(* IEC 61131-3 sources: CodesysTest/export/Function Blocks/SolenoidValves/FB_PneumaticActuator.pou/RetractAsserted.prop, 1 file *)

(* ---- Get.pm.st ---- *)
(*#-#-#-#-#-#-#-#-#-#---Declaration---#-#-#-#-#-#-#-#-#-#-#-#-#*)

VAR
END_VAR
(*#-#-#-#-#-#-#-#-#-#---Implementation---#-#-#-#-#-#-#-#-#-#-#-#-#*)

RetractAsserted := _retractAsserted;
